{attribute 'GeneratedUsingTerminal: ELX9410-0000-0016'}
{attribute addProperty BoxType "ELX9410-0000-0016"}
{attribute addProperty Id "EtcSlaveTerminalBaseStatus_UsAT %I*Status_Us_B1E819A21Status_UpAT %I*Status_Up_B1E819A21WcStateAT %I*WcState_9091E0EB2InfoDataAT %I*InfoData_6F19DB2B2"}
{attribute addProperty CRC "229053890"}
{attribute addProperty Size "6"}
TYPE ELX9410_0DA715C2 EXTENDS EtcSlaveTerminalBase :
STRUCT
	{attribute addProperty Name "Status_Us"}
	Status_Us : Status_Us_B1E819A2;
	{attribute addProperty Name "Status_Up"}
	Status_Up : Status_Up_B1E819A2;
	{attribute addProperty Name "WcState"}
	WcState : WcState_9091E0EB;
	{attribute addProperty Name "InfoData"}
	InfoData : InfoData_6F19DB2B;
END_STRUCT
END_TYPE

(* stored: Version 1.2.0.0, ProductVersion 3.1.4024.9
   DUT ELX9410_0DA715C2: Id {c1e872c2-139e-4894-b368-4a108a43115e} *)
